(* Schneider Machine Expert - Basic project New project, file version 2.7.0.0 *)
(* ProjectInformations: Name=New project *)

HARDWARE
  Cpu 0: TM200C24R
  EthernetConfiguration: NetworkName=M200, IpAllocationMode=FixedAddress, IpAddress=0.0.0.0, SubnetMask=0.0.0.0
  SerialLineConfiguration: Baud=Baud19200, Parity=ParityEven, DataBits=DataBits8, StopBits=StopBits1, PhysicalMedium=PhysicalMediumRs485, TransmissionMode=TransmissionModeModbusRtu, SlaveId=1, Addressing=SlaveAddressing
  MastTask: UsePeriodScanMode=false, PeriodScan=100
  FastTask: Period=255
  CpuBehavior: StartingMode=StartAsPreviousState, AutoSaveRamOnEeprom=true, WatchdogPeriod=250

SYMBOLS  (address, symbol, comment, settings)

POU New POU
  (* SectionNumber=1 *)

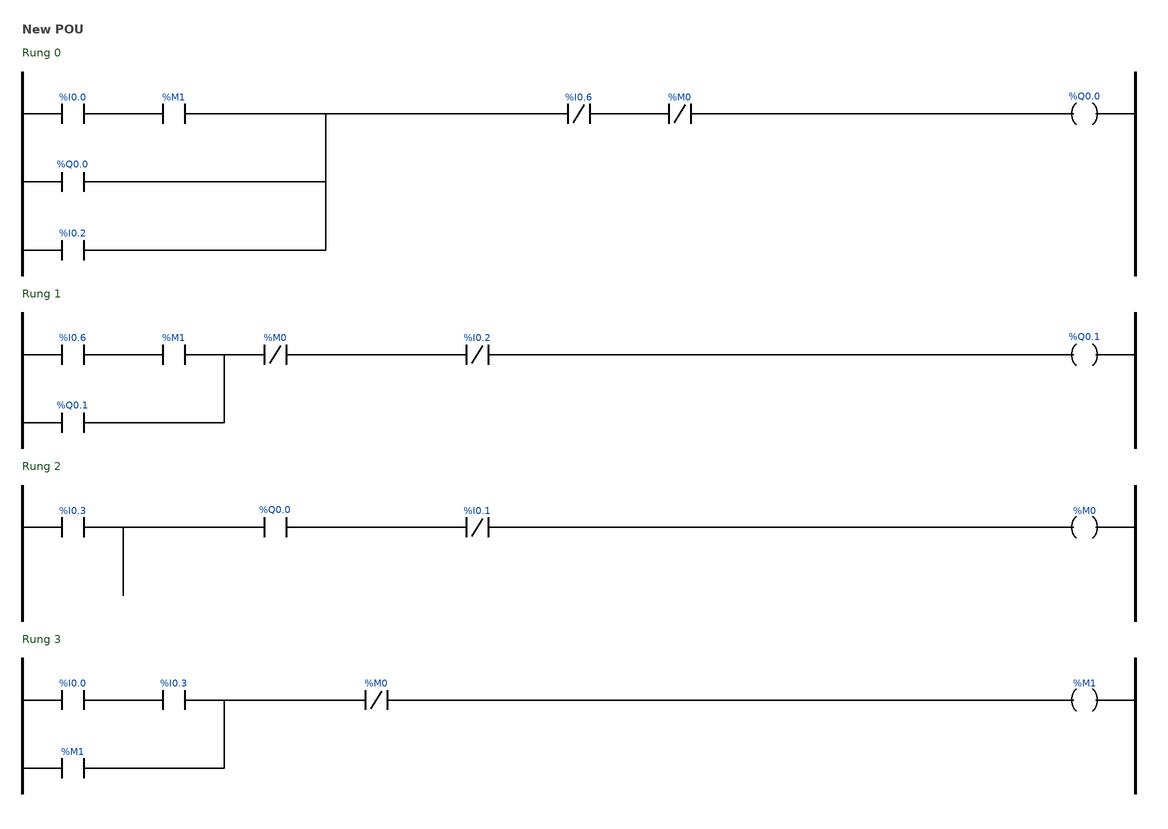

// Rung 0
  LD %I0.0
  AND %M1
  OR %Q0.0
  OR %I0.2
  ANDN %I0.6
  ANDN %M0
  ST %Q0.0
  // as ST:
  //   %Q0.0 := (%I0.0 AND %M1 OR %Q0.0 OR %I0.2) AND NOT %I0.6 AND NOT %M0;

// Rung 1
  LD %I0.6
  AND %M1
  OR %Q0.1
  ANDN %M0
  ANDN %I0.2
  ST %Q0.1
  // as ST:
  //   %Q0.1 := (%I0.6 AND %M1 OR %Q0.1) AND NOT %M0 AND NOT %I0.2;

// Rung 2
  (* no IL stored for this rung *)

// Rung 3
  LD %I0.0
  AND %I0.3
  OR %M1
  ANDN %M0
  ST %M1
  // as ST:
  //   %M1 := (%I0.0 AND %I0.3 OR %M1) AND NOT %M0;
